{attribute addProperty BoxType "ELX9560-0000-0016"}
{attribute addProperty Id "Status_UinAT %I*Status_Uin_324A4102810Status_UexAT %I*Status_Uex_324A4102810WcStateAT %I*WcState_F855686C1620InfoDataAT %I*InfoData_192954DE1620"}
{attribute addProperty CRC "2892798250"}
{attribute addProperty SizeInBites "48"}
{attribute addProperty SizeInBytes "6"}
TYPE ELX9560_FB68D8D1 :
STRUCT
	{attribute addProperty Name "Status_Uin"}
	Status_Uin : Status_Uin_324A4102;
	{attribute addProperty Name "Status_Uex"}
	Status_Uex : Status_Uex_324A4102;
	{attribute addProperty Name "WcState"}
	WcState : WcState_F855686C;
	{attribute addProperty Name "InfoData"}
	InfoData : InfoData_192954DE;
END_STRUCT
END_TYPE

(* stored: Version 1.2.0.0, ProductVersion 3.1.4024.9
   DUT ELX9560_FB68D8D1: Id {5b77c298-4dff-4c4b-858b-57129841935f} *)
